//{attribute 'qualified_only'}
VAR_GLOBAL

    (*HXR Accelerator side PLC Interface*)
    Accelerator_Upstream_Gauge	:	ST_VG;

    {attribute 'TcLinkTo' :=	'TIIB[EBD_E5_EL1008]^Channel 1^Input
    '}
    i_xUpstreamTreaty_PressOK	AT	%I*	:	BOOL;
//	{attribute 'TcLinkTo' :=	'TIIB[EBD_E8_EL2794]^Channel 1^Output
//	'}
//	q_xUpstreamTreaty_PressOK	AT	%Q*	:	BOOL;


    (*HXR Gas Attenuator PLC Interface*)

    fb_ADS_WATCHDOG_VAC_LFE_GEM:FB_ADS_WATCHDOG;

    (*TXI PLC Interface*)
	{attribute 'TcLinkTo' := 	'.i_rPRESS	:=	TIIB[TXI_HXR_VAC_PLC (EL6692)]^IO Inputs^PC2L1_PIP_01_rPress;
								.i_xAT_VAC	:=	TIIB[TXI_HXR_VAC_PLC (EL6692)]^IO Inputs^PC2L1_PIP_01_AT_VAC;
								.i_xPRESS_OK	:=	TIIB[TXI_HXR_VAC_PLC (EL6692)]^IO Inputs^PC2L1_PIP_01_PRESS_OK
	
    '}
	PC2L1_L2SI_PIP_01:FB_Gauge_Interface;
    (*XPP PLC Interface*)
    {attribute 'pytmc' := '
            pv: PLC:LFE:VAC:XPP:DS:GCC_EPICS
    '}
    XPP_Downstream_Gauge		:	ST_VG;
    XPP_Modbus_Gauge		:	FB_GaugeModbus; //ST_VG;
    XPP_DS_Gauge		:	ST_VG;


    {attribute 'pytmc' := '
            pv: PLC:LFE:VAC:XPP:Downstream:PMON
            link: HX3:MON:GCC:01:PMON
    '}
    XPP_PressureLinkHelper : FB_LREALFromEPICS;

END_VAR

(* stored: Version 1.1.0.1, ProductVersion 3.1.4022.18
   GVL GVL_PLC_Interfaces: Id {fcddf43e-c4e4-4dff-b9ca-620efda50799} *)
